// TIA Portal V16 export
// export: Created 2022-09-01T14:26:58.6926078Z, ExportSetting WithDefaults, DisplayName Totally Integrated Automation Portal, DisplayVersion V16, DisplayName TIA Portal Version Control Interface, DisplayVersion V16, DisplayName TIA Portal Openness, DisplayVersion V16, DisplayName STEP 7 Professional, DisplayVersion V16, DisplayName STEP 7 Safety, DisplayVersion V16, DisplayName WinCC Advanced, DisplayVersion V16
FUNCTION "Controlo_Pressostatos" : Void   // FC8, LAD
TITLE = Ao fim de 30s indica que atingiu setpoint de pressão
{ S7_Optimized_Access := 'TRUE' }
VERSION : 0.1
// stored: AutoNumber true, IsIECCheckEnabled false, SetENOAutomatically false, UDAEnableTagReadback false
BEGIN

REGION Network 1: Pressostato Filtro 1
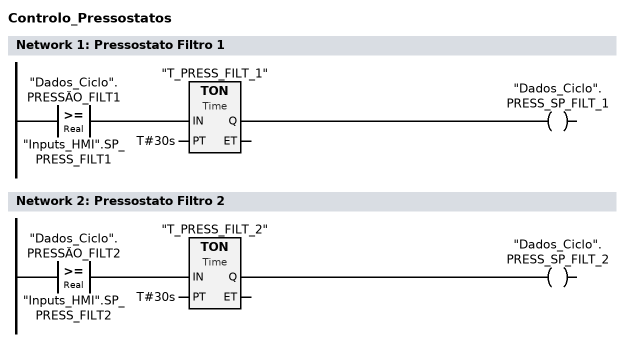
   RUNG wire#powerrail
      { S7_Templates := "SrcType := Real" } GE_Contact(in1 := "Dados_Ciclo".PRESSÃO_FILT1, in2 := "Inputs_HMI".SP_PRESS_FILT1)
      { S7_Templates := "time_type := Time" } "T_PRESS_FILT_1".TON(pt := T#30s, et =>)
      Coil( "Dados_Ciclo".PRESS_SP_FILT_1 )
   END_RUNG
   // the same network as SCL:
   "T_PRESS_FILT_1".TON(IN := "Dados_Ciclo".PRESSÃO_FILT1 >= "Inputs_HMI".SP_PRESS_FILT1, PT := T#30s);
   "Dados_Ciclo".PRESS_SP_FILT_1 := "T_PRESS_FILT_1".Q;
END_REGION

REGION Network 2: Pressostato Filtro 2
   RUNG wire#powerrail
      { S7_Templates := "SrcType := Real" } GE_Contact(in1 := "Dados_Ciclo".PRESSÃO_FILT2, in2 := "Inputs_HMI".SP_PRESS_FILT2)
      { S7_Templates := "time_type := Time" } "T_PRESS_FILT_2".TON(pt := T#30s, et =>)
      Coil( "Dados_Ciclo".PRESS_SP_FILT_2 )
   END_RUNG
   // the same network as SCL:
   "T_PRESS_FILT_2".TON(IN := "Dados_Ciclo".PRESSÃO_FILT2 >= "Inputs_HMI".SP_PRESS_FILT2, PT := T#30s);
   "Dados_Ciclo".PRESS_SP_FILT_2 := "T_PRESS_FILT_2".Q;
END_REGION
END_FUNCTION
